{attribute 'GeneratedUsingTerminal: EL3443-0000-0017'}
{attribute addProperty BoxType "EL3443-0000-0017"}
{attribute addProperty Id "L1_StatusAT %I*L1_Status_61BE889610L1_BasicAT %I*L1_Basic_665874DE8L1_PowerAT %I*L1_Power_22301EDD16L1_TimingAT %I*L1_Timing_CCFF711F8L2_StatusAT %I*L2_Status_61BE889610L2_BasicAT %I*L2_Basic_665874DE8L2_PowerAT %I*L2_Power_22301EDD16L2_TimingAT %I*L2_Timing_CCFF711F8L3_StatusAT %I*L3_Status_61BE889610L3_BasicAT %I*L3_Basic_665874DE8L3_PowerAT %I*L3_Power_22301EDD16L3_TimingAT %I*L3_Timing_CCFF711F8Total_StatusAT %I*Total_Status_1ACE98F018Total_BasicAT %I*Total_Basic_FC2CFF1712Total_ActiveAT %I*Total_Active_F9B49EA128Total_Total_L_L_VoltageAT %I*Total_Total_L_L_Voltage_2881351912WcStateAT %I*WcState_9091E0EB2InfoDataAT %I*InfoData_94A18F5E2"}
{attribute addProperty CRC "3419666542"}
{attribute addProperty Size "200"}
TYPE EL3443_CBD3F86E EXTENDS EtcSlaveTerminalBase_947E5A46 :
STRUCT
	{attribute addProperty Name "L1_Status"}
	L1_Status : L1_Status_61BE8896;
	{attribute addProperty Name "L1_Basic"}
	L1_Basic : L1_Basic_665874DE;
	{attribute addProperty Name "L1_Power"}
	L1_Power : L1_Power_22301EDD;
	{attribute addProperty Name "L1_Timing"}
	L1_Timing : L1_Timing_CCFF711F;
	{attribute addProperty Name "L2_Status"}
	L2_Status : L2_Status_61BE8896;
	{attribute addProperty Name "L2_Basic"}
	L2_Basic : L2_Basic_665874DE;
	{attribute addProperty Name "L2_Power"}
	L2_Power : L2_Power_22301EDD;
	{attribute addProperty Name "L2_Timing"}
	L2_Timing : L2_Timing_CCFF711F;
	{attribute addProperty Name "L3_Status"}
	L3_Status : L3_Status_61BE8896;
	{attribute addProperty Name "L3_Basic"}
	L3_Basic : L3_Basic_665874DE;
	{attribute addProperty Name "L3_Power"}
	L3_Power : L3_Power_22301EDD;
	{attribute addProperty Name "L3_Timing"}
	L3_Timing : L3_Timing_CCFF711F;
	{attribute addProperty Name "Total_Status"}
	Total_Status : Total_Status_1ACE98F0;
	{attribute addProperty Name "Total_Basic"}
	Total_Basic : Total_Basic_FC2CFF17;
	{attribute addProperty Name "Total_Active"}
	Total_Active : Total_Active_F9B49EA1;
	{attribute addProperty Name "Total_Total_L_L_Voltage"}
	Total_Total_L_L_Voltage : Total_Total_L_L_Voltage_28813519;
	{attribute addProperty Name "WcState"}
	WcState : WcState_9091E0EB;
	{attribute addProperty Name "InfoData"}
	InfoData : InfoData_94A18F5E;
END_STRUCT
END_TYPE

(* stored: Version 1.2.0.0, ProductVersion 3.1.4024.9
   DUT EL3443_CBD3F86E: Id {7ba9605b-4ac6-44c4-8d82-b3a32d0820b3} *)
